// TIA Portal V16 program export: 2 tag tables, 0 data types, 0 data blocks, 3 code blocks (in call order from the OBs), 1 instance data blocks

VAR_GLOBAL   // PLC tag table "Standard-Variablentabelle"
   Clock_Byte AT %MB1 : Byte;
   Clock_10Hz AT %M1.0 : Bool;
   Clock_5Hz AT %M1.1 : Bool;
   "Clock_2.5Hz" AT %M1.2 : Bool;
   Clock_2Hz AT %M1.3 : Bool;
   "Clock_1.25Hz" AT %M1.4 : Bool;
   Clock_1Hz AT %M1.5 : Bool;
   "Clock_0.625Hz" AT %M1.6 : Bool;
   "Clock_0.5Hz" AT %M1.7 : Bool;
   "Reset Coutner" AT %I2.0 : Bool;
   "Reset Coutner Light" AT %Q1.4 : Bool;
END_VAR

VAR_GLOBAL   // PLC tag table "Tag table from XML_1"
   "Moving X" AT %I0.0 : Bool;
   "Moving Z" AT %I0.1 : Bool;
   "Item detected" AT %I0.2 : Bool;
   "Lid at place" AT %I0.3 : Bool;
   "Lid clamped" AT %I0.4 : Bool;
   "Pos. at limit (lids)" AT %I0.5 : Bool;
   "Base at place" AT %I0.6 : Bool;
   "Base clamped" AT %I0.7 : Bool;
   "Pos. at limit (bases)" AT %I1.0 : Bool;
   "Part leaving" AT %I1.1 : Bool;
   Start AT %I1.2 : Bool;
   Reset AT %I1.3 : Bool;
   Stop AT %I1.4 : Bool;
   "Emergency stop" AT %I1.5 : Bool;
   Auto AT %I1.6 : Bool;
   "FACTORY I/O (Uruchomiony)" AT %I1.7 : Bool;
   "Move X" AT %Q0.0 : Bool;
   "Move Z" AT %Q0.1 : Bool;
   Grab AT %Q0.2 : Bool;
   "Lids conveyor" AT %Q0.3 : Bool;
   "Clamp lid" AT %Q0.4 : Bool;
   "Pos. raise (lids)" AT %Q0.5 : Bool;
   "Bases conveyor" AT %Q0.6 : Bool;
   "Clamp base" AT %Q0.7 : Bool;
   "Pos. raise (bases)" AT %Q1.0 : Bool;
   "Start light" AT %Q1.1 : Bool;
   "Reset light" AT %Q1.2 : Bool;
   "Stop light" AT %Q1.3 : Bool;
   "Counter" AT %QD30 : DInt;
END_VAR

ORGANIZATION_BLOCK "Main"   // OB1, LAD, ProgramCycle
TITLE = "Main Program Sweep (Cycle)"
{ S7_Optimized_Access := 'TRUE' }
VERSION : 0.1
// stored: AutoNumber true, IsIECCheckEnabled false, SetENOAutomatically false
   VAR_INPUT
      Initial_Call : Bool;   // Initial call of this OB
      Remanence : Bool;   // =True, if remanent data are available
   END_VAR
   VAR_TEMP
      temp : Real;
   END_VAR
BEGIN

REGION Network 1
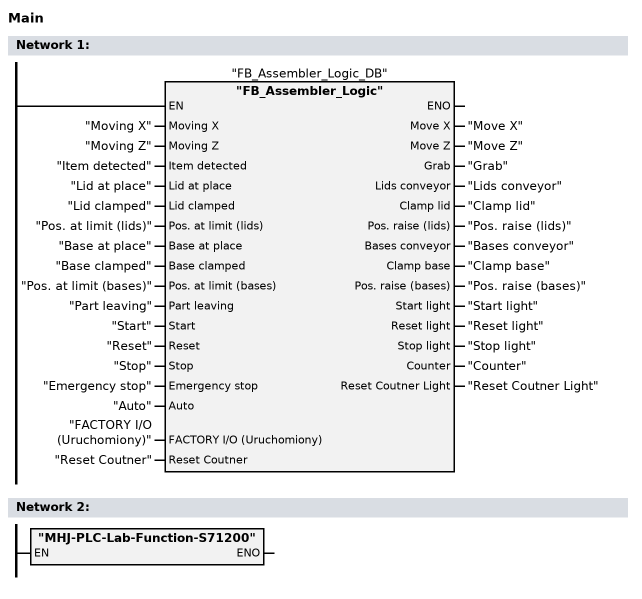
   RUNG wire#powerrail
      "FB_Assembler_Logic_DB"("Moving X" := "Moving X", "Moving Z" := "Moving Z", "Item detected" := "Item detected", "Lid at place" := "Lid at place", "Lid clamped" := "Lid clamped", "Pos. at limit (lids)" := "Pos. at limit (lids)", "Base at place" := "Base at place", "Base clamped" := "Base clamped", "Pos. at limit (bases)" := "Pos. at limit (bases)", "Part leaving" := "Part leaving", Start := "Start", Reset := "Reset", Stop := "Stop", "Emergency stop" := "Emergency stop", Auto := "Auto", "FACTORY I/O (Uruchomiony)" := "FACTORY I/O (Uruchomiony)", "Reset Coutner" := "Reset Coutner", "Move X" => "Move X", "Move Z" => "Move Z", Grab => "Grab", "Lids conveyor" => "Lids conveyor", "Clamp lid" => "Clamp lid", "Pos. raise (lids)" => "Pos. raise (lids)", "Bases conveyor" => "Bases conveyor", "Clamp base" => "Clamp base", "Pos. raise (bases)" => "Pos. raise (bases)", "Start light" => "Start light", "Reset light" => "Reset light", "Stop light" => "Stop light", "Counter" => "Counter", "Reset Coutner Light" => "Reset Coutner Light")
   END_RUNG
   // the same network as SCL:
   "FB_Assembler_Logic_DB"("Moving X" := "Moving X",   // "FB_Assembler_Logic"
                           "Moving Z" := "Moving Z",
                           "Item detected" := "Item detected",
                           "Lid at place" := "Lid at place",
                           "Lid clamped" := "Lid clamped",
                           "Pos. at limit (lids)" := "Pos. at limit (lids)",
                           "Base at place" := "Base at place",
                           "Base clamped" := "Base clamped",
                           "Pos. at limit (bases)" := "Pos. at limit (bases)",
                           "Part leaving" := "Part leaving",
                           Start := "Start",
                           Reset := "Reset",
                           Stop := "Stop",
                           "Emergency stop" := "Emergency stop",
                           Auto := "Auto",
                           "FACTORY I/O (Uruchomiony)" := "FACTORY I/O (Uruchomiony)",
                           "Reset Coutner" := "Reset Coutner",
                           "Move X" => "Move X",
                           "Move Z" => "Move Z",
                           Grab => "Grab",
                           "Lids conveyor" => "Lids conveyor",
                           "Clamp lid" => "Clamp lid",
                           "Pos. raise (lids)" => "Pos. raise (lids)",
                           "Bases conveyor" => "Bases conveyor",
                           "Clamp base" => "Clamp base",
                           "Pos. raise (bases)" => "Pos. raise (bases)",
                           "Start light" => "Start light",
                           "Reset light" => "Reset light",
                           "Stop light" => "Stop light",
                           "Counter" => "Counter",
                           "Reset Coutner Light" => "Reset Coutner Light");
END_REGION

REGION Network 2
   RUNG wire#powerrail
      "MHJ-PLC-Lab-Function-S71200"()
   END_RUNG
   // the same network as SCL:
   "MHJ-PLC-Lab-Function-S71200"();
END_REGION
END_ORGANIZATION_BLOCK

FUNCTION_BLOCK "FB_Assembler_Logic"
{ S7_Optimized_Access := 'TRUE' }
VERSION : 0.1
   VAR_INPUT 
      "Moving X" : Bool;
      "Moving Z" : Bool;
      "Item detected" : Bool;
      "Lid at place" : Bool;
      "Lid clamped" : Bool;
      "Pos. at limit (lids)" : Bool;
      "Base at place" : Bool;
      "Base clamped" : Bool;
      "Pos. at limit (bases)" : Bool;
      "Part leaving" : Bool;
      Start : Bool;
      Reset : Bool;
      Stop : Bool;
      "Emergency stop" : Bool;
      Auto : Bool;
      "FACTORY I/O (Uruchomiony)" : Bool;
      "Reset Coutner" : Bool;
   END_VAR

   VAR_OUTPUT 
      "Move X" : Bool;
      "Move Z" : Bool;
      Grab : Bool;
      "Lids conveyor" : Bool;
      "Clamp lid" : Bool;
      "Pos. raise (lids)" : Bool;
      "Bases conveyor" : Bool;
      "Clamp base" : Bool;
      "Pos. raise (bases)" : Bool;
      "Start light" : Bool;
      "Reset light" : Bool;
      "Stop light" : Bool;
      "Counter" : DInt;
      "Reset Coutner Light" : Bool;
   END_VAR

   VAR 
      stat_Step : Int;
      stat_TrigLid {InstructionName := 'F_TRIG'; LibVersion := '1.0'; S7_SetPoint := 'False'} : F_TRIG;
      stat_TrigBase {InstructionName := 'F_TRIG'; LibVersion := '1.0'} : F_TRIG;
      stat_LidDone { S7_SetPoint := 'True'} : Bool;
      stat_BaseDone : Bool;
      timerLift {InstructionName := 'TON_TIME'; LibVersion := '1.0'; S7_SetPoint := 'False'} : TON_TIME;
      stat_HoldingPart { S7_SetPoint := 'True'} : Bool;
      stat_X_Started : Bool;
      stat_Z_Started : Bool;
      System_Pracuje : Bool;
      Awaria_Aktywna : Bool;
   END_VAR


BEGIN
	// --- 1. LOGIKA PAMIĘCI AWARII (LATCH) ---
	// Jeśli wciśnięto E-Stop, ustawiamy stan awarii.
	// Stan ten trwa nawet po wyciśnięciu E-Stop, aż do naciśnięcia Reset.
	IF NOT #"Emergency stop" THEN
	    #Awaria_Aktywna := TRUE;
	END_IF;
	
	IF #Reset AND #"Emergency stop" THEN
	   #Awaria_Aktywna := FALSE;  // Kasowanie awarii tylko gdy grzybek jest wyciśnięty 
	END_IF;
	
	// --- 2. LOGIKA PRACY (START/STOP) ---
	// System może pracować tylko gdy nie ma aktywnej awarii
	IF #"Start" AND NOT #Awaria_Aktywna AND #"Stop" AND #"Emergency stop" THEN
	    #System_Pracuje := TRUE;
	ELSIF NOT #"Stop"  OR #Awaria_Aktywna THEN
	    #System_Pracuje := FALSE;
	END_IF;
	
	// --- 3. STEROWANIE LAMPKAMI ---
	// Lampka RESET
	IF #Awaria_Aktywna THEN
	    #"Reset light" :="Clock_1Hz";  // Miga dopóki nie wciśniesz Reset
	ELSE
	    #"Reset light":= FALSE;
	END_IF;
	
	// Lampka START (zielona)
	IF #System_Pracuje THEN
	    #"Start light" := TRUE;        // Pali się ciągle podczas pracy
	ELSIF NOT #Awaria_Aktywna AND #"Emergency stop" AND #Stop THEN
	    #"Start light" := "Clock_1Hz";  // Miga po Resecie (gotowość do Startu)
	ELSE
	    #"Start light" := FALSE;       // Ciemna podczas awarii
	END_IF;
	
	// Lampka STOP (czerwona)
	IF NOT #System_Pracuje THEN
	    #"Stop light" := TRUE;
	ELSE
	    #"Stop light" := FALSE;
	END_IF;
	// Reset Coutnera
	IF #"Reset Coutner" THEN
	    #"Reset Coutner Light" := TRUE;
	    #"Counter" := 0;
	ELSE
	    #"Reset Coutner Light" := FALSE;
	END_IF;
	    
	// --- 4. AUTOMAT STANÓW (GŁÓWNY PROCES) ---
	// Sterowanie procesem tylko gdy system pracuje
	IF #System_Pracuje THEN
	    CASE #stat_Step OF
	            
	        0:  // TRANSPORT ELEMENTÓW ZA CZUJNIKI (NC + R_TRIG)
	            #stat_TrigLid(CLK := #"Lid at place");
	            #stat_TrigBase(CLK := #"Base at place");
	            
	            // Jeśli element mija czujnik NC (powrót sygnału na 1), zatrzymaj taśmę
	            IF #stat_TrigLid.Q THEN
	                #stat_LidDone := TRUE;
	            END_IF;
	            IF #stat_TrigBase.Q THEN
	                #stat_BaseDone := TRUE;
	            END_IF;
	            
	            #"Lids conveyor" := NOT #stat_LidDone;
	            #"Bases conveyor" := NOT #stat_BaseDone;
	            
	            IF #stat_LidDone AND #stat_BaseDone THEN
	                #stat_LidDone := FALSE;
	                #stat_BaseDone := FALSE;
	                #stat_Step := 10;
	            END_IF;
	            
	        10: // ZACISKANIE (Zaciski NC: zaciśnięte = FALSE)
	            #"Clamp lid" := TRUE;
	            #"Clamp base" := TRUE;
	            IF NOT #"Lid clamped" AND NOT #"Base clamped" THEN
	                #stat_Step := 20;
	            END_IF;
	            
	        20: // MOVE Z (Zjazd w dół po pokrywę)
	            #"Move Z" := TRUE;
	            IF NOT #"Moving Z" AND #"Item detected" THEN
	                #stat_Step := 30;
	            END_IF;
	            
	        30: // GRAB & PODNIESIENIE (Zjazd Z w górę)
	            #stat_HoldingPart := TRUE;  // Chwytak ON (podtrzymany globalnie)
	            #"Move Z" := FALSE;            // Komenda: Jedź w górę
	            #"Clamp lid" := FALSE;         // Puść zacisk pokrywy
	            
	            // Czekaj aż ramię dotrze na górę i ustabilizuje element
	            #timerLift(IN := (NOT #"Moving Z" AND #"Item detected"),
	                       PT := T#100ms);
	            
	            IF #timerLift.Q THEN
	                #stat_Step := 40;
	            END_IF;
	            
	        40: // MOVE X (Przejazd w osi X nad podstawę)
	            #timerLift(IN := FALSE,
	                       PT := T#100ms); // Reset timera z poprzedniego kroku
	            
	            #"Move X" := TRUE; // Uruchomienie ruchu
	            
	            // LOGIKA PRZEJŚCIA:
	            // Musimy mieć pewność, że ruch wystartował (Moving X = TRUE)
	            // a następnie zakończył się (Moving X = FALSE)
	            IF #"Move X" AND NOT #"Moving X" AND #stat_X_Started THEN
	                #stat_X_Started := FALSE; // Reset flagi pomocniczej
	                #stat_Step := 50;
	            END_IF;
	            
	            // Flaga pomocnicza wykrywająca, że ramię ruszyło
	            IF #"Moving X" THEN
	                #stat_X_Started := TRUE;
	            END_IF;
	            
	        50: // MOVE Z (Opuszczenie pokrywy na podstawę)
	            #"Move Z":= TRUE;
	            
	            // Czekaj na koniec ruchu osi Z w dół
	            IF #"Move Z" AND NOT #"Moving Z" AND #stat_Z_Started THEN
	                #stat_Z_Started := FALSE;
	                #stat_Step := 60;
	            END_IF;
	            IF #"Moving Z" THEN
	                #stat_Z_Started := TRUE;
	            END_IF;
	            
	        60: // GRAB OFF (Puszczenie elementu)
	            #stat_HoldingPart := FALSE; // Chwytak OFF
	            #"Move Z" := FALSE;
	            
	            // Czekaj aż czujnik potwierdzi, że element odpadł od chwytaka
	            IF NOT #"Item detected" THEN
	                #stat_Step := 70;
	            END_IF;
	            
	        70: // POWRÓT RAMIENIA I WYPUŚCZENIE PRODUKTU
	            #"Move Z" := FALSE;
	            #"Move X" := FALSE;
	            #"Clamp base" := FALSE; // Puść gotowy produkt
	            
	            // 1. Czekaj na powrót ramienia, aby bezpiecznie podnieść transporter
	            IF NOT #"Moving X" AND NOT #"Moving Z" THEN
	                #"Pos. raise (bases)" := TRUE;
	                #"Bases conveyor":= TRUE;
	            END_IF;
	            
	            // 2. Gdy produkt zacznie opuszczać stację (wejście na czujnik Part leaving)
	            IF #"Part leaving" THEN
	                #"Pos. raise (bases)" := FALSE; // Opuść blokadę
	                #Counter := #Counter + 1;   // Naliczenie sztuki
	                #stat_Step := 80;           // Przejdź do kroku oczekiwania na odjazd
	            END_IF;
	            
	        80: // OCZEKIWANIE NA CAŁKOWITY ODJAZD (Stabilizacja licznika)
	            // Czekamy, aż produkt całkowicie zniknie z czujnika (dla NC sygnał wróci na TRUE)
	            // Zapobiega to wielokrotnemu naliczeniu tej samej sztuki
	            IF #"Part leaving"THEN
	                #stat_Step := 0;
	            END_IF;
	            
	    END_CASE;
	    
	ELSE
	    // Awaryjne wyłączenie wszystkich napędów
	    #"Lids conveyor" := FALSE;
	    #"Bases conveyor" := FALSE;
	    #"Move X":= FALSE;
	    #"Move Z":= FALSE;
	    #"Clamp lid":= FALSE;
	    #"Clamp base" := FALSE;
	    #stat_HoldingPart := FALSE;
	END_IF;
	
	// --- 5. PODTRZYMANIE SYGNAŁU CHWYTAKA ---
	// Podtrzymanie sygnału Grab niezależnie od kroku, aby robot nie upuszczał części
	#Grab := #stat_HoldingPart;
	
	// --- 6. RESET FLAG POMOCNICZYCH I TIMERÓW ---
	// Reset flag i timerów przy zatrzymaniu systemu
	IF NOT #System_Pracuje THEN
	    #stat_Step := 0;
	    #stat_HoldingPart := FALSE;
	    
	    #stat_X_Started := FALSE;  // Czyścimy pamięć ruchu X
	    #stat_Z_Started := FALSE;  // Czyścimy pamięć ruchu Z
	    
	    // Reset timera, aby nie "wisiały" przy ponownym starcie
	    #timerLift(IN := FALSE,
	               PT := T#100ms);
	END_IF;
	
END_FUNCTION_BLOCK

FUNCTION "MHJ-PLC-Lab-Function-S71200" : Void
{ S7_Optimized_Access := 'TRUE' }
VERSION : 0.1
   VAR_TEMP 
      rdTimeReturn : Int;
      outputTime {InstructionName := 'DTL'; LibVersion := '1.0'} : DTL;
      SyncVal : Byte;
      forVal : Int;
      forVal_2 : Int;
      Value : Byte;
   END_VAR

   VAR CONSTANT 
      CompVal : Byte := 16#34;
      Value_01 : Byte := 16#11;
      Value_01_DW : DWord := 16#A165_D992;
      Value_02_DW : DWord := 16#58BE_4401;
   END_VAR


BEGIN
	
	#Value:=PEEK(area := 16#82,
	     dbNumber := 0,
	     byteOffset := 511);
	#Value := #Value + 1;
	
	POKE(area := 16#82,
	     dbNumber := 0,
	     byteOffset := 511,
	     value := #Value);
	
	POKE(area:=16#81,
	     dbNumber:=0,
	     byteOffset:=1016,
	     value:=#Value_01_DW);
	POKE(area := 16#81,
	     dbNumber := 0,
	     byteOffset := 1020,
	     value := #Value_02_DW);
	
	POKE(area := 16#81,
	     dbNumber := 0,
	     byteOffset := 511,
	     value := B#16#00);
	
	FOR #forVal := 0 TO 120 DO
	    FOR #forVal_2:=0 TO 10 DO
	        #rdTimeReturn:=RD_SYS_T(#outputTime);
	        #rdTimeReturn := WR_SYS_T(#outputTime);
	        #rdTimeReturn := RD_SYS_T(#outputTime);
	        #rdTimeReturn := WR_SYS_T(#outputTime);
	    END_FOR;
	    #SyncVal:= PEEK(area := 16#81,
	                   dbNumber := 0,
	                   byteOffset := 511);
	    IF #SyncVal = #CompVal THEN
	       GOTO M_1;
	    END_IF;
	END_FOR;
	RETURN;
	
	M_1:
	POKE(area := 16#81,
	     dbNumber := 0,
	     byteOffset := 511,
	     value := B#16#0);
	
	
	    
END_FUNCTION

DATA_BLOCK "FB_Assembler_Logic_DB"   // DB1
VERSION : 0.1
// stored: AutoNumber true, InstanceOfName FB_Assembler_Logic, InstanceOfType FB
"FB_Assembler_Logic"
BEGIN
END_DATA_BLOCK
